{attribute 'GeneratedUsingTerminal: EL7332-0000-0016'}
{attribute addProperty BoxType "EL7332-0000-0016"}
{attribute addProperty Id "DCM_Status_Channel_1AT %I*DCM_Status_Channel_36ED096F11DCM_Status_Channel_2AT %I*DCM_Status_Channel_36ED096F11DCM_Control_Channel_1AT %Q*DCM_Control_Channel_5A8B50163DCM_Velocity_Channel_1AT %Q*DCM_Velocity_Channel_A47A3F412DCM_Control_Channel_2AT %Q*DCM_Control_Channel_5A8B50163DCM_Velocity_Channel_2AT %Q*DCM_Velocity_Channel_A47A3F412WcStateAT %I*WcState_9091E0EB2InfoDataAT %I*InfoData_3B4F4E8A4"}
{attribute addProperty CRC "3095768317"}
{attribute addProperty Size "38"}
TYPE EL7332_B885ACFD EXTENDS EtcSlaveTerminalBase_947E5A46 :
STRUCT
	{attribute addProperty Name "DCM_Status_Channel_1"}
	DCM_Status_Channel_1 : DCM_Status_Channel_36ED096F;
	{attribute addProperty Name "DCM_Status_Channel_2"}
	DCM_Status_Channel_2 : DCM_Status_Channel_36ED096F;
	{attribute addProperty Name "DCM_Control_Channel_1"}
	DCM_Control_Channel_1 : DCM_Control_Channel_5A8B5016;
	{attribute addProperty Name "DCM_Velocity_Channel_1"}
	DCM_Velocity_Channel_1 : DCM_Velocity_Channel_A47A3F41;
	{attribute addProperty Name "DCM_Control_Channel_2"}
	DCM_Control_Channel_2 : DCM_Control_Channel_5A8B5016;
	{attribute addProperty Name "DCM_Velocity_Channel_2"}
	DCM_Velocity_Channel_2 : DCM_Velocity_Channel_A47A3F41;
	{attribute addProperty Name "WcState"}
	WcState : WcState_9091E0EB;
	{attribute addProperty Name "InfoData"}
	InfoData : InfoData_3B4F4E8A;
END_STRUCT
END_TYPE

(* stored: Version 1.2.0.0, ProductVersion 3.1.4024.9
   DUT EL7332_B885ACFD: Id {4e1553c6-10ab-4121-9fa9-9c9eade5db3a} *)
